SUBAPPLICATION Uebung_020d (* DigitalInput_I1 auf DigitalOutput_Q1; TOF Ausschaltverzögert *)
  (* Standard: 61499-2 *)
  (* Version 1.0, 2023-10-23, franz *)
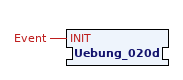
  EVENT_INPUT
    INIT;
  END_EVENT
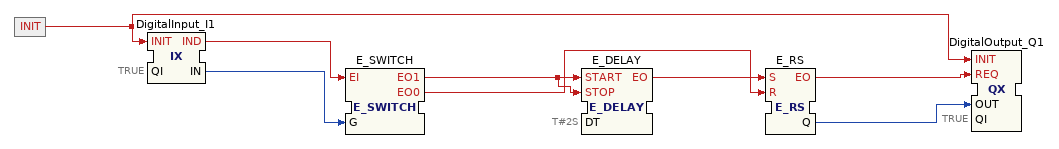
  FBS
    DigitalOutput_Q1 : QX(QI := TRUE);
    DigitalInput_I1 : IX(QI := TRUE);
    E_SWITCH : E_SWITCH;
    E_RS : E_RS;
    E_DELAY : E_DELAY(DT := T#2S);
  END_FBS
  EVENT_CONNECTIONS
    INIT TO DigitalInput_I1.INIT;
    INIT TO DigitalOutput_Q1.INIT;
    DigitalInput_I1.IND TO E_SWITCH.EI;
    E_RS.EO TO DigitalOutput_Q1.REQ;
    E_SWITCH.EO1 TO E_RS.S;
    E_SWITCH.EO0 TO E_DELAY.START;
    E_DELAY.EO TO E_RS.R;
    E_SWITCH.EO1 TO E_DELAY.STOP;
  END_CONNECTIONS
  DATA_CONNECTIONS
    DigitalInput_I1.IN TO E_SWITCH.G;
    E_RS.Q TO DigitalOutput_Q1.OUT;
  END_CONNECTIONS
END_SUBAPPLICATION
